Staubli VAL3: Edit.pgx

program Edit()
  local bool l_bRes
  local num l_i
  local string l_sValue
  local num l_nSelect
  local string l_sItem
  local num l_nKey
  local num l_nRes
begin

  cls()
  resize(sParameter,1,6)
  sParameter[0]="X"
  sParameter[1]="Y"
  sParameter[2]="Z"
  sParameter[3]="Rx"
  sParameter[4]="Ry"
  sParameter[5]="Rz"
  //
  resize(sListItemValue,1,size(sParameter))
  sListItemValue[0]=toString(".3",fFrame[sItem].trsf.x)
  sListItemValue[1]=toString(".3",fFrame[sItem].trsf.y)
  sListItemValue[2]=toString(".3",fFrame[sItem].trsf.z)
  sListItemValue[3]=toString(".3",fFrame[sItem].trsf.rx)
  sListItemValue[4]=toString(".3",fFrame[sItem].trsf.ry)
  sListItemValue[5]=toString(".3",fFrame[sItem].trsf.rz)
  //
  for l_i=0 to size(sParameter)-1
    call user:strlength(sParameter[l_i],user:nBottomX/2)
    l_sValue=sListItemValue[l_i]
    call user:strlength(l_sValue,user:nBottomX/2+1)
    sParameter[l_i]=sParameter[l_i]+":"+l_sValue
  endFor

  bUserRefresh=true
  bListRefresh=true
  //
  do
    if bUserRefresh
      cls()
      call user:clear(0,13)
      call user:typeMenu(8,"确定")
    endIf
    call user:setList(sItem,sParameter,bUserRefresh,bListRefresh,l_nSelect,l_sItem,l_nKey)
    bUserRefresh=false
    bListRefresh=false
    call EnterPageKey(l_nKey,l_nSelect,sParameter[l_nSelect])
    delay(0)
  until l_nKey==255 or l_nKey==278
  bUserRefresh=true
  bListRefresh=true
end
